TYPE TcoDatamanConfig_v_5_x_x :
STRUCT
	ReadDataLength : UINT := 246;
	UserDataLength : UINT := 252;
END_STRUCT
END_TYPE

(* stored: Version 1.1.0.1, ProductVersion 3.1.4024.11
   DUT TcoDatamanConfig_v_5_x_x: Id {511d8c94-eb01-0087-0253-264e18e831b8} *)
